Omron CX-Programmer project NewProject (CX-Programmer 9.73)

# PLC NewPLC1: CP1E N20

## Global symbols (name address type ; comment)
0.01 BOOL  ; SENSOR
0.03 BOOL  ; RESET
100.00 BOOL  ; LAMPU
100.04 BOOL  ; OUTPUT
C001 BOOL  ; COUNTER
T002 BOOL  ; TIMER

## Program NewProgram1 (cyclic task 0)

### Section Section1

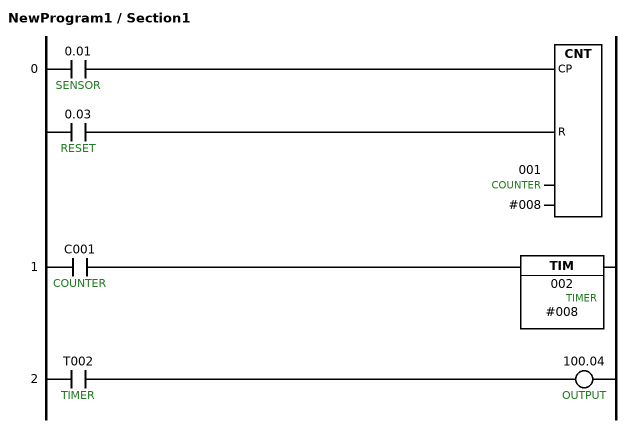
; rung 0
LD 0.01  ; SENSOR
LD 0.03  ; RESET
CNT 001 #008  ; COUNTER
; rung 1
LD C001  ; COUNTER
TIM 002 #008  ; TIMER
; rung 2
LD T002  ; TIMER
OUT 100.04  ; OUTPUT

### Section END
; rung 0
END(001)